// TIA Portal project "第三节课上升沿和下降沿" (V15.1)

(* hardware
DEVICE "S7-1200 station_1"  S7-1200 Station
   slot 0: "Rack_0"  S7-1200 Rack  Rack  V1.0
   slot 1: "PLC_1"  CPU 1212C DC/DC/DC  6ES7 212-1AE40-0XB0  V4.2
*)

// ===== PLC "PLC_1"  CPU 1212C DC/DC/DC =====

VAR_GLOBAL   // PLC tag table "变量表_1"
   "总开关" AT %I0.4 : Bool;
   "保护开关" AT %I0.5 : Bool;
   "输出(1)" AT %Q0.1 : Bool;
   "电机启动" AT %M0.5 : Bool;
   "电机关闭" AT %M0.6 : Bool;
   "电机启动1" AT %M0.7 : Bool;
   "电机关闭1" AT %M1.0 : Bool;
END_VAR

VAR_GLOBAL   // PLC tag table "io"
   "上升" AT %I0.0 : Bool;
   "下降" AT %I0.1 : Bool;
   "输出" AT %Q0.0 : Bool;
   "中间扫描1" AT %M0.1 : Bool;
   "中间扫描2" AT %M0.2 : Bool;
   "上升1" AT %I0.2 : Bool;
   "下降1" AT %I0.3 : Bool;
   "中间扫描3" AT %M0.3 : Bool;
   "中间扫描4" AT %M0.4 : Bool;
   "中间数值" AT %MW100 : Word;
END_VAR

ORGANIZATION_BLOCK "Main"   // OB1, LAD, ProgramCycle
TITLE = "Main Program Sweep (Cycle)"
{ S7_Optimized_Access := 'TRUE' }
VERSION : 0.1
   VAR_INPUT
      Initial_Call : Bool;   // Initial call of this OB
      Remanence : Bool;   // =True, if remanent data are available
   END_VAR
   VAR_TEMP   // added for the SCL form of the ladder/FBD networks
      _w1 : Bool;
      _w2 : Bool;
   END_VAR
BEGIN

REGION Network 1
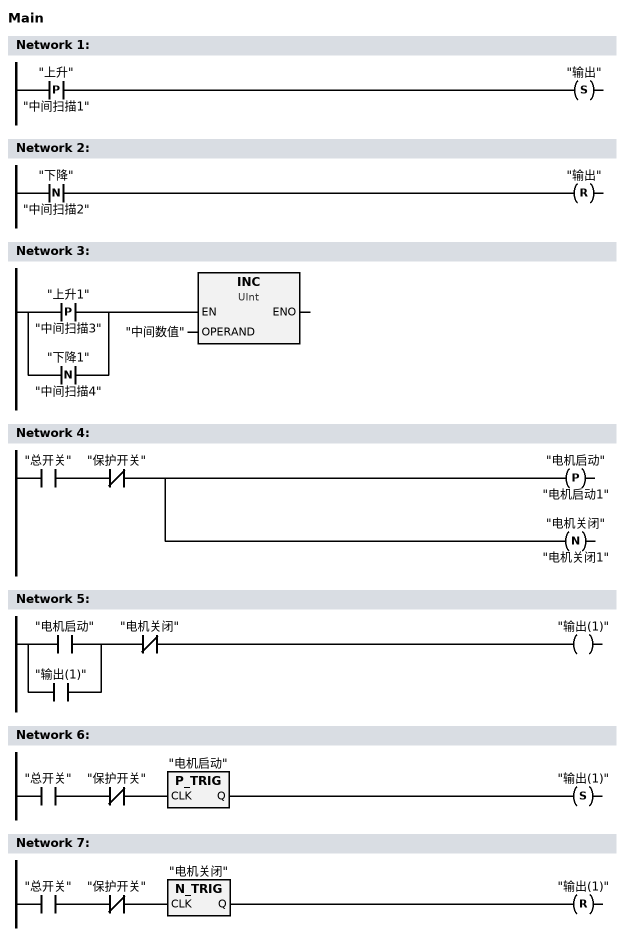
   RUNG wire#powerrail
      P_Contact(operand := "上升", bit := "中间扫描1")
      S_Coil( "输出" )
   END_RUNG
   // the same network as SCL:
   #_w1 := "上升" AND NOT "中间扫描1";   // rising edge of "上升"
   "中间扫描1" := "上升";
   IF #_w1 THEN "输出" := TRUE; END_IF;
END_REGION

REGION Network 2
   RUNG wire#powerrail
      N_Contact(operand := "下降", bit := "中间扫描2")
      R_Coil( "输出" )
   END_RUNG
   // the same network as SCL:
   #_w1 := NOT "下降" AND "中间扫描2";   // falling edge of "下降"
   "中间扫描2" := "下降";
   IF #_w1 THEN "输出" := FALSE; END_IF;
END_REGION

REGION Network 3
   RUNG wire#powerrail
      P_Contact(operand := "上升1", bit := "中间扫描3")
      wire#w1
      { S7_Templates := "DestType := UInt" } Inc( "中间数值" )
   END_RUNG
   RUNG wire#powerrail
      N_Contact(operand := "下降1", bit := "中间扫描4")
   END_RUNG wire#w1
   // the same network as SCL:
   #_w1 := "上升1" AND NOT "中间扫描3";   // rising edge of "上升1"
   "中间扫描3" := "上升1";
   #_w2 := NOT "下降1" AND "中间扫描4";   // falling edge of "下降1"
   "中间扫描4" := "下降1";
   IF #_w1 OR #_w2 THEN "中间数值" := "中间数值" + 1; END_IF;
END_REGION

REGION Network 4
   #_w1 := "总开关" AND NOT "保护开关";
   "电机启动" := #_w1 AND NOT "电机启动1";   // rising edge
   "电机启动1" := #_w1;
   "电机关闭" := NOT #_w1 AND "电机关闭1";   // falling edge
   "电机关闭1" := #_w1;
END_REGION

REGION Network 5
   RUNG wire#powerrail
      Contact( "电机启动" )
      wire#w1
      I_Contact( "电机关闭" )
      Coil( "输出(1)" )
   END_RUNG
   RUNG wire#powerrail
      Contact( "输出(1)" )
   END_RUNG wire#w1
   // the same network as SCL:
   "输出(1)" := ("电机启动" OR "输出(1)") AND NOT "电机关闭";
END_REGION

REGION Network 6
   RUNG wire#powerrail
      Contact( "总开关" )
      I_Contact( "保护开关" )
      P_Trig( "电机启动" )
      S_Coil( "输出(1)" )
   END_RUNG
   // the same network as SCL:
   #_w1 := "总开关" AND NOT "保护开关";
   #_w2 := #_w1 AND NOT "电机启动";   // rising edge
   "电机启动" := #_w1;
   IF #_w2 THEN "输出(1)" := TRUE; END_IF;
END_REGION

REGION Network 7
   RUNG wire#powerrail
      Contact( "总开关" )
      I_Contact( "保护开关" )
      N_Trig( "电机关闭" )
      R_Coil( "输出(1)" )
   END_RUNG
   // the same network as SCL:
   #_w1 := "总开关" AND NOT "保护开关";
   #_w2 := NOT #_w1 AND "电机关闭";   // falling edge
   "电机关闭" := #_w1;
   IF #_w2 THEN "输出(1)" := FALSE; END_IF;
END_REGION
END_ORGANIZATION_BLOCK